FUNCTION_BLOCK CPress (* Composite Function Block Type *)
  (* Standard: 61499-2 *)
  (* Version 0.0, 30/03/2026, template *)
  PACKAGE Hidryco.HidrycoLib;
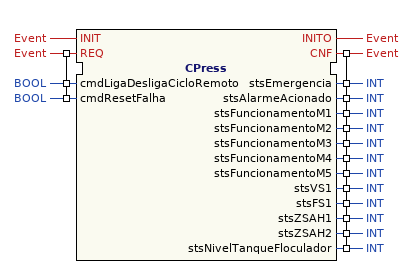
  EVENT_INPUT
    INIT; (* Initialization Request *)
    REQ WITH cmdLigaDesligaCicloRemoto, cmdResetFalha; (* Normal Execution Request *)
  END_EVENT
  EVENT_OUTPUT
    INITO; (* Initialization Confirm *)
    CNF WITH stsEmergencia, stsAlarmeAcionado, stsFuncionamentoM1, stsFuncionamentoM2, stsFuncionamentoM3, stsFuncionamentoM4, stsFuncionamentoM5, stsVS1, stsFS1, stsZSAH1, stsZSAH2, stsNivelTanqueFloculador; (* Execution Confirmation *)
  END_EVENT
  VAR_INPUT
    cmdLigaDesligaCicloRemoto : BOOL;
    cmdResetFalha : BOOL;
  END_VAR
  VAR_OUTPUT
    stsEmergencia : INT;
    stsAlarmeAcionado : INT; (* Alarme H *)
    stsFuncionamentoM1 : INT; (* Funcionamento da prensa M1. *)
    stsFuncionamentoM2 : INT; (* Funcionamento do moto redutor limpeza M2 *)
    stsFuncionamentoM3 : INT; (* Funcionamento do agitador floculador M3 *)
    stsFuncionamentoM4 : INT; (* Funcionamento da bomba de água M4 *)
    stsFuncionamentoM5 : INT; (* Funcionamento do compressor M5 *)
    stsVS1 : INT; (* Status da válvula solenoide de limpeza VS1 *)
    stsFS1 : INT; (* Status chave de fluxo FS1 *)
    stsZSAH1 : INT; (* Fim de curso frontal limpeza ZSAH1 *)
    stsZSAH2 : INT; (* Fim de curso trazeira limpeza ZSAH2 *)
    stsNivelTanqueFloculador : INT;
  END_VAR
  FBS
    SYMLINKMULTIVARSRC1 : SYMLINKMULTIVARSRC_277E97BEC1451D2C(NAME1 := '$${PATH}cmdLigaDesligaCicloRemoto', NAME2 := '$${PATH}cmdResetFalha', QI := TRUE); {SET_ATTRIBUTE(Configuration.GenericFBType.InterfaceParams, Runtime.System#I:=2;VALUE${I$}:BOOL,BOOL)}
    SYMLINKMULTIVARDST1 : SYMLINKMULTIVARDST_182274139AA51730B(NAME1 := '$${PATH}stsEmergencia', NAME2 := '$${PATH}stsAlarmeAcionado', NAME3 := '$${PATH}stsFuncionamentoM1', NAME4 := '$${PATH}stsFuncionamentoM2', NAME5 := '$${PATH}stsFuncionamentoM3', NAME6 := '$${PATH}stsFuncionamentoM4', NAME7 := '$${PATH}stsFuncionamentoM5', NAME8 := '$${PATH}stsVS1', NAME9 := '$${PATH}stsFS1', NAME10 := '$${PATH}stsZSAH1', NAME11 := '$${PATH}stsZSAH2', NAME12 := '$${PATH}stsNivelTanqueFloculador', QI := TRUE); {SET_ATTRIBUTE(Configuration.GenericFBType.InterfaceParams, Runtime.System#I:=12;VALUE${I$}:INT,INT,INT,INT,INT,INT,INT,INT,INT,INT,INT,INT)}
    IThis : CPress_HMI(QI := TRUE);
  END_FBS
  EVENT_CONNECTIONS
    REQ TO SYMLINKMULTIVARSRC1.REQ;
    SYMLINKMULTIVARDST1.CNF TO CNF;
    INIT TO SYMLINKMULTIVARSRC1.INIT;
    SYMLINKMULTIVARSRC1.INITO TO SYMLINKMULTIVARDST1.INIT;
    SYMLINKMULTIVARDST1.INITO TO IThis.64521A07ED789434;
    SYMLINKMULTIVARDST1.CNF TO IThis.A8B8B70E79878008;
    IThis.899D2916F7D03DF6 TO INITO;
  END_CONNECTIONS
  DATA_CONNECTIONS
    SYMLINKMULTIVARDST1.VALUE1 TO stsEmergencia;
    SYMLINKMULTIVARDST1.VALUE2 TO stsAlarmeAcionado;
    SYMLINKMULTIVARDST1.VALUE3 TO stsFuncionamentoM1;
    SYMLINKMULTIVARDST1.VALUE4 TO stsFuncionamentoM2;
    SYMLINKMULTIVARDST1.VALUE5 TO stsFuncionamentoM3;
    SYMLINKMULTIVARDST1.VALUE6 TO stsFuncionamentoM4;
    SYMLINKMULTIVARDST1.VALUE7 TO stsFuncionamentoM5;
    SYMLINKMULTIVARDST1.VALUE8 TO stsVS1;
    SYMLINKMULTIVARDST1.VALUE9 TO stsFS1;
    SYMLINKMULTIVARDST1.VALUE10 TO stsZSAH1;
    SYMLINKMULTIVARDST1.VALUE11 TO stsZSAH2;
    SYMLINKMULTIVARDST1.VALUE12 TO stsNivelTanqueFloculador;
    cmdLigaDesligaCicloRemoto TO SYMLINKMULTIVARSRC1.VALUE1;
    cmdResetFalha TO SYMLINKMULTIVARSRC1.VALUE2;
    SYMLINKMULTIVARDST1.VALUE1 TO IThis.64D3B0F867C0D9E6;
    SYMLINKMULTIVARDST1.VALUE2 TO IThis.169B62C9497170F5;
    SYMLINKMULTIVARDST1.VALUE3 TO IThis.E4933AC304504E98;
    SYMLINKMULTIVARDST1.VALUE4 TO IThis.D3E0284FD4C0DAB8;
    SYMLINKMULTIVARDST1.VALUE5 TO IThis.8679CF31D8003532;
    SYMLINKMULTIVARDST1.VALUE6 TO IThis.4810B5E36EF99D65;
    SYMLINKMULTIVARDST1.VALUE7 TO IThis.3B99ADC4C179ABEE;
    SYMLINKMULTIVARDST1.VALUE8 TO IThis.FF36CEC9C61030EB;
    SYMLINKMULTIVARDST1.VALUE9 TO IThis.9F191C5490979C1D;
    SYMLINKMULTIVARDST1.VALUE10 TO IThis.26C74165CA13B157;
    SYMLINKMULTIVARDST1.VALUE11 TO IThis.702DC38A923F5BDD;
    SYMLINKMULTIVARDST1.VALUE12 TO IThis.44371829128A4C3D;
  END_CONNECTIONS
END_FUNCTION_BLOCK
